PROGRAM P_Demo_FB_DALIV2QueryControlGearPresent
VAR
    fbFB_DALIV2QueryControlGearPresent        : FB_DALIV2QueryControlGearPresent;
    stCommandBuffer : ST_DALIV2CommandBuffer;

    bTrigger        : BOOL;
    nLampAddr        : BYTE := 0;

    bResult          : BOOL;

    bBusy           : BOOL;
    bErr            : BOOL;
    nErrId          : UDINT;
END_VAR

// =============================================================================
// 场景：巡检 short addr 0：查询灯具是否在线（应答 = 在线）。
//
// 价值：HMI 显示用。
//
// 验证步骤：
//   1. 通信 FB 跑起；编译；登录。
//   2. 在线 bTrigger 一次上升沿；等 bBusy 回 FALSE。
//   3. 观察 fbFB_DALIV2QueryControlGearPresent.bQueryData 应为预期值（参考本 FB 文档 §4 描述）。
// =============================================================================
fbFB_DALIV2QueryControlGearPresent(
    bStart           := bTrigger,
    nAddr            := nLampAddr,
    eAddrType        := eDALIV2AddrTypeShort,
    eCommandPriority := eDALIV2CommandPriorityLow,
    stCommandBuffer  := stCommandBuffer
);

bBusy  := fbFB_DALIV2QueryControlGearPresent.bBusy;
bErr   := fbFB_DALIV2QueryControlGearPresent.bError;
nErrId := fbFB_DALIV2QueryControlGearPresent.nErrorId;

END_PROGRAM

(* stored: Version 1.1.0.1, ProductVersion 3.1.4024.5
   POU P_Demo_FB_DALIV2QueryControlGearPresent: Id {2705b28a-5cf6-5bd5-bf8e-89bf168e2985}, SpecialFunc None *)
